PROGRAM MAIN
VAR
	nCounter : INT := 10_000; 
END_VAR

END_PROGRAM

(* stored: Version 1.1.0.1, ProductVersion 3.1.4024.9
   POU MAIN: Id {f2c55725-7b8a-4083-abeb-dc6829ffb8f1}, SpecialFunc None *)
